{attribute 'qualified_only'}
VAR_GLOBAL
	stMainStateMachine				: ST_MainStateMachineHmi;
END_VAR

(* stored: Version 1.1.0.1, ProductVersion 3.1.4024.11
   GVL Hmi: Id {c01be153-0ad2-49c4-8fdf-7f8869731658} *)
